(*

.. <legal notes>

legal notes
=================
| SPDX-FileCopyrightText: © 2026 Oleksandr Tiutyk <trofimich@gmail.com>
| SPDX-License-Identifier: LGPL-3.0-only
| For details check: LGPL-3.0-only_

.. _LGPL-3.0-only: https://www.gnu.org/licenses/lgpl-3.0.en.html

.. </legal notes>

*)

INTERFACE IAutomationController EXTENDS IParentAutomationComponent

{attribute 'monitoring' := 'call'}
PROPERTY FINAL PluginCount : Core.INT_LENGTH
GET
END_GET
END_PROPERTY

METHOD TryGetPluginByIndex : IAutomationControllerPlugin
VAR_INPUT
	index : Core.INT_INDEX;
END_VAR
END_METHOD

END_INTERFACE

(* stored: Version 1.1.0.1
   Itf IAutomationController: Id {0b4e8e80-e173-49c5-86a2-54e893b4c200}
   Property PluginCount: Id {b6aa27af-1d06-4aea-8e2c-3eda3657bf33}
   Get Get: Id {a7f23203-43c8-446f-82f0-3a72173748c8}
   Method TryGetPluginByIndex: Id {ba60eef3-9279-4fda-8f5e-7bace35abbbc} *)
